PROGRAM MAIN_load_arch
VAR
	vector_2 : ARRAY[0..4] OF LREAL := [1,1,1,1,1];	
	out : ARRAY[0..0] OF LREAL;
	FB_NN : FB_Dense_v1;
	
	runtime_profiler : PROFILER;
	profiler_data : PROFILERSTRUCT;
	
	buf_idx : UINT := 0;
	profiler_buffer : ARRAY [0..1000] OF DWORD;
	
	MeasureFinished : BOOL := TRUE;

	

END_VAR


runtime_profiler(START := TRUE, RESET := TRUE);
FB_NN(pointer_input := ADR(vector_2),pointer_output:= ADR(out));

runtime_profiler(START := FALSE);
profiler_data := runtime_profiler.DATA;
IF NOT MeasureFinished THEN
	profiler_buffer[buf_idx] := profiler_data.LastExecTime;
	buf_idx := buf_idx+1; 
	buf_idx := buf_idx MOD (SIZEOF(profiler_buffer)/SIZEOF(DWORD)); // len of profiler_buffer
	IF buf_idx = 0 THEN
		MeasureFinished := TRUE;
	END_IF
END_IF


//sum := F_DATA_TO_CRC16_CCITT(pData := ADR(FB_NN.nn.weights),cbData := SIZEOF(FB_NN.nn.weights),crc:=crc);
//sum2 := F_CheckSum16(dwSrcAddr := ADR(FB_NN.nn.weights),cbLen := SIZEOF(FB_NN.nn.weights),wChkSum:=crc);

END_PROGRAM

(* stored: Version 1.1.0.1, ProductVersion 3.1.4024.12
   POU MAIN_load_arch: Id {37181db8-c75f-4678-aa7c-0dd71cdd5322}, SpecialFunc None *)
